TYPE CAGroupInfo :
STRUCT
	sName 		: STRING;
	nId			: OTCID;
	eGroupState	: MC_GROUP_STATE;
	nAxesCount 	: INT; 
END_STRUCT
END_TYPE

(* stored: Version 1.1.0.1
   DUT CAGroupInfo: Id {77fbe3b9-8052-450c-bbca-6778d31915fb} *)
